// TwinCAT 3 PLC project Untitled1
// ProgramVersion: 3.1.4024.0
// libraries:
//   Tc2_Math, * (Beckhoff Automation GmbH)
//   Tc2_Standard, * (Beckhoff Automation GmbH)
//   Tc2_System, * (Beckhoff Automation GmbH)
//   Tc2_Utilities, * (Beckhoff Automation GmbH)
//   Tc3_Mc3PlanarMotion, * (Beckhoff Automation GmbH)
//   Tc3_Module, * (Beckhoff Automation GmbH)
//   Tc3_Physics, * (Beckhoff Automation GmbH)
//   Tc3_XPlanarUtility, * (Beckhoff Automation GmbH & Co. KG)
//   XboxControllerUtilities, * (Beckhoff Community)
// project tree:
//   DUTs/ Motion_Parameters.TcDUT, Environment_Parameters.TcDUT
//   / PlcTask.TcTTO
//   POUs/Controller/ XboxController.TcPOU
//   POUs/Demo/ Demo.TcPOU
//   POUs/Enviorment/ Environment.TcPOU
//   POUs/ MAIN.TcPOU
//   POUs/Xplanar/Mover Type/ AMP4220.TcPOU, AMP4330.TcPOU
//   POUs/Xplanar/ XPlanarMover.TcPOU
// real-time tasks:
//   TASK Job Task: cycle default, priority 13
//   TASK PlcTask: cycle T#250us, priority 10, ADS port 350
//   TASK XPlanar Task3: cycle T#250us, priority 4, ADS port 351
//   TASK XPlanar Task4: cycle T#250us, priority 6, ADS port 352
//   TASK MC-Task (MET): cycle T#250us, priority 8, ADS port 353
//   TASK MC-Task (MPT): cycle T#10ms, priority 14, ADS port 354
// variable links:
//   XPlanar MC Project/Axes/Mover4220_1 <-> TcCOM Objects/XPlanar/Mover4220_1
//     McToIo/STD <-> InputsFromNC3/NC3ToHW
//   Untitled1/Untitled1 Instance <-> XPlanar MC Project/Axes/Mover4220_1
//     PlcTask Inputs/MAIN.MyMover.Xplanar_Mover.MCTOPLC/ACT <-> McToPlc/ACT
//     PlcTask Inputs/MAIN.MyMover.Xplanar_Mover.MCTOPLC/COORDMODE <-> McToPlc/COORDMODE
//     PlcTask Inputs/MAIN.MyMover.Xplanar_Mover.MCTOPLC/SET <-> McToPlc/SET
//     PlcTask Inputs/MAIN.MyMover.Xplanar_Mover.MCTOPLC/SETONTRACK <-> McToPlc/SETONTRACK
//     PlcTask Inputs/MAIN.MyMover.Xplanar_Mover.MCTOPLC/STD <-> McToPlc/STD
//     PlcTask Outputs/MAIN.MyMover.Xplanar_Mover.PLCTOMC/STD <-> PlcToMc/STD
//   TcCOM Objects/XPlanar/Mover4220_1 <-> XPlanar MC Project/Axes/Mover4220_1
//     OutputsToNC3/HWToNC3 <-> IoToMc/STD

CONFIGURATION Untitled1
    RESOURCE PLC ON TwinCAT3
        TASK PlcTask(INTERVAL := T#250us, PRIORITY := 10);
        PROGRAM MAIN WITH PlcTask : MAIN;
    END_RESOURCE
END_CONFIGURATION

// ---- DUTs/Motion_Parameters.TcDUT
TYPE Motion_Parameters :
STRUCT
	
	
			maxAcceleration					: 		LREAL	:= 15000;			// mm/s^2
		
			maxVelocity						: 		LREAL	:= 500.0;			// mm/s
		
			minVelocity						: 		LREAL	:= -500.0;			// -mm/s
		
			RotationScailing				: 		LREAL 	:= 0.0005; 			// Radians/s^2
		
			CenteringFactor					:		LREAL	:= 0.002;			// Radians/s^2
		
			tiltscailing					:  		LREAL 	:= 0.008; 			// scailing from controller to radians 

END_STRUCT
END_TYPE

// ---- DUTs/Environment_Parameters.TcDUT
TYPE Environment_Parameters :
STRUCT
	
			Friction_coefficient			:  		LREAL 	:= 9.50 ; 			// Frictiton of table
			
			deltaT							:		LREAL	:= 0.00025;			//Cycle time 

END_STRUCT
END_TYPE

// ---- POUs/MAIN.TcPOU
PROGRAM MAIN
VAR
	
MyMover : XplanarMover; // Xplanar Mover

MyController : XboxController; // Xbox Controller

MyEnvironment : Environment; // Xplanar Environment

MyDemo : Demo; // Xplanar Demo 

END_VAR
























VAR
	bRumble : BOOL;  // Set rumble true for haptics based on conditions
END_VAR

Cyclic(); 


MyMover(
// Part number of mover being controlled	
MoverType := 'AMP4220',
Space_Mode := FALSE //Fun time - need to reactivate if set true or false 
); 

MyController(
// Set true if you want haptics and false if you dont	
HapticFeedback := TRUE
);

MyEnvironment(
// Input number of X and Y tiles youre table has
NumberOfXTiles := 4, 
NumberOfYTiles := 3	
);

ACTION Cyclic:
Haptics();

//Initizalization
MyMover.Init( 
bStart := MyController.Start,
Reinit := MyDemo.StartUserControl
);

//Recover 
MyMover.Recover(
bBack := MyController.Reset
); 

//tilt
MyMover.Tilt_Height(
rStick_X := MyController.rStick_X,
rStick_Y := MyController.rStick_Y,
bButton_B := MyController.Button_B,
LBumper := MyController.lBumper,
RBumper	:= MyController.rBumper
);

//X and Y Movement 
MyMover.XYMovement(
lStick_X := MyController.lStick_X, 
lStick_Y := MyController.lStick_Y, 
bButton_A := MyController.Button_A, 
bButton_X := MyController.Button_X, 
bButton_Y := MyController.Button_Y, 
maxXTravel := MyEnvironment.MaxTableXTravel,
minXTravel := MyEnvironment.MinTableXTravel,
maxYTravel := MyEnvironment.MaxTableYTravel,
minYTravel := MyEnvironment.MinTableYTravel,

);

MyMover.Rotation(
LTrigger := MyController.lTrigger,
RTrigger := MyController.rTrigger
);

MyController.takeScreenshot(
bDpad_D := Mycontroller.Dpad_D,
MoverPosition := MyMover.Xplanar_Mover.MCTOPLC.ACT.ActPos
);

MyController.clearScreenshot(
bDpad_U := MyController.Dpad_U,
ClearPosition := MyController.ZeroVector
);

MyController.Haptics(
Rumble := bRumble,
BackTo0Rumble := MyMover.RotationRumble
);

MyEnvironment.Boundry(
MoverTypeWidth 				:= MyMover.TypeWidth, 
MoverTypeLength				:= MyMover.TypeLength 
);

MyMover(
StartDemo := MyDemo.RequestDemo,
DemoNotReady :=  MyDemo.StartUserControl
); 


MyDemo(
ReadyForDemo := MyMover.DemoReady,
bDpad_R := MyController.Dpad_R,
bDpad_L := MyController.Dpad_L,
StopEndFunction := MyMover.ResetDemo,
DemoTable := MyEnvironment.TableType,
//Running := MyMover.FourByThree.Running OR MyMover.TwoByOne.Running,
//Done := MyMover.FourByThree.Done OR MyMover.TwoByOne.Done
);

MyMover.FourByThree(
Start:= MyDemo.StartFourByThree,
Stop := MyDemo.StopFourByThree
);

MyMover.TwoByOne(
Start:= MyDemo.StartTwoByOne,
Stop := MyDemo.StopTwoByOne
);




MyMover(); 
MyController();
MyEnvironment();
MyDemo();
END_ACTION

METHOD Haptics
VAR_INPUT
END_VAR
VAR_OUTPUT
END_VAR
VAR
END_VAR
//When found a rotation point or at a boundry 
IF NOT MyMover.Space_mode THEN // IF space mode is on chnage the way table detection is done
	IF (MyController.Button_A AND MyMover.RotationXPoint AND MyMover.RotationYPoint) 
	OR (MyController.lBumper OR MyController.rBumper) 
	OR ((MyEnvironment.MinTableXTravel + 1 > MyMover.PlanarMoverPos.X) 
	OR (MyEnvironment.MinTableYTravel + 1 > MyMover.PlanarMoverPos.Y) 
	OR (MyEnvironment.MaxTableYTravel - 1 < MyMover.PlanarMoverPos.Y) 
	OR (MyEnvironment.MaxTableXTravel - 1 < MyMover.PlanarMoverPos.X))THEN
		bRumble := TRUE;
	ELSE
		bRumble := FALSE;
	END_IF
ELSE
	//Increase mover detection on boundry
	IF (MyController.Button_A AND MyMover.RotationXPoint AND MyMover.RotationYPoint) 
	OR (MyController.lBumper OR MyController.rBumper) 
	OR (((MyEnvironment.MinTableXTravel + 15) > MyMover.PlanarMoverPos.X) 
	OR ((MyEnvironment.MinTableYTravel + 15) > MyMover.PlanarMoverPos.Y) 
	OR ((MyEnvironment.MaxTableYTravel - 15) < MyMover.PlanarMoverPos.Y) 
	OR ((MyEnvironment.MaxTableXTravel - 15) < MyMover.PlanarMoverPos.X))THEN
		bRumble := TRUE;
	ELSE
		bRumble := FALSE;
	END_IF
END_IF
END_METHOD

END_PROGRAM

// ---- POUs/Xplanar/XPlanarMover.TcPOU
FUNCTION_BLOCK XPlanarMover
VAR_INPUT
	
			MotionParameters			:		Motion_Parameters; // Min-max Motion parameters

			MoverType					: 		STRING(7); //Input what mover is being controlled
			
			Space_mode					:		BOOL; // Space mode ???
			
			StartDemo					:		BOOL; // Change to Demo
			DemoNotReady 				: 		BOOL; //Handeling for end process

END_VAR
VAR_OUTPUT
	
			Xplanar_Mover 				: 		MC_PlanarMover; // Xplanr Mover fb
			moverState					:		MC_Planar_State; // State of mover
			
			TypeWidth					: 		LREAL; //Mover Width  		
			TypeLength					:		LREAL; //Mover Length
			
			PlanarMoverPos				:		MoverVector; // Haptic Handeling
			
			RotationXPoint				:		BOOL; // At rotation point for haptics
			RotationYPoint				:		BOOL; // At rotation point for haptics
			RotationRumble				:		BOOL; // At 0 output for haptics
			
			DemoReady					:		BOOL; // Handshake to start demo
			ResetDemo					:		BOOL; // Hnadshake to stop end demo
			
END_VAR
VAR
	
			stExtOptions				:		ARRAY [1..2]  OF ST_ExternalSetpointGenerationOptions; // External Setpoint options
			cmdFB 						:		ARRAY [1..2]  OF MC_PlanarFeedBack ; //Mover Feedback 
			XpPosition					:		MoverVector; // Commanded mover pos
			MoverPos					:		MoverVector; // Act pos of mover
			ZeroVector 					:		MoverVector; // Zero feed for External Pos

			
			
			EnvironmentParameters		:		Environment_Parameters; // Enviroment parameters like table boundry, fricition coeffecent 
			typeAMP4220					: 		AMP4220; // Mover 4220 decleration	
			typeAMP4330					:		AMP4330; // Mover 4330 decleration
			
		
			//Init Vars
			Run 						:		BOOL; // Run init case	
			DONE						: 		BOOL; // Done running init
			nCase 						: 		SINT := 1; // Case of init
			init_counter				:		INT; // How many times we can try to recover

			
 			//X Y vars
			SumnedForce_X				: 		LREAL; // Calculation of applied force on X
			SumnedForce_Y 				: 		LREAL; // Calculation of applied force on Y
			Mover_acceleration			: 		MoverVector; // Commanded Mover Acc
			friction_force				: 		MoverVector; // Fricition against mover
			SumnedVelocity				: 		MoverVector; // Commanded Velocity after intergation 
			
			
			//Recover Vars
			nRecover					:		SINT := 1; // Case of Recover
			bRecover					: 		BOOL; // Recover mover 
			
			
			//Height Vars
			Height 						: 		LREAL := 2; // Varible in which height is passed
			Left_OSR					: 		R_TRIG; // OSR to make sure a left bumper click is counted a one
			Right_OSR					: 		R_TRIG; // OSR to make sure a right bumper click is counted a one
			Left_Bumer_TON				:		TON; // Timer for incremental lowering 
			Right_Bumper_TON			:		TON; // Timer for incremental rising 
			Smoothing_Left_TON			:		TON; // Timer for smoothing on lowering 
			Smoothing_Right_TON			:		TON; // Timer for smoothing on rising 
			
			//Tilt Vars
			Holding_Contact				:		BOOL; // Holding bool for Button B
			Release_Contact				:		BOOL; // Release bool for holding contact
			Button_B_OSR				: 		R_TRIG; // OSR to make sure a Button B click is counted a one
			nButton						:		INT := 1; // Case for holding contact
			
			//Rotation Vars
			DestinationX				: 		DINT; // Rotation point on X plane
			DestinationY				: 		DINT; // Rotation point on Y plane 
			AtXPoint					: 		BOOL; // At x point on table 
			AtYPoint					: 		BOOL; // At Y point on table 
			MaxPosRot					: 		LREAL; // Max Positive rotation allowed if not at rotation point
			MaxNegRot					: 		LREAL; // Max Negative rotation allowed if not at rotation point
			isintent					: 		BOOL; // mChecking to see if mover is standstill
			Closest90					:		LREAL; // Finding the closest position that is moduled by 90 from actual pos
			MODDED_C					: 		INT; // Modded C value for math check
			PastRot10					: 		BOOL; // Past +- 01 degress check
			Centering_Direction			:		SINT; // Check to see which direction mover needs to center in
			LowerBound 					: 		LREAL; // Lower bound of Centering position
			UpperBound 					: 		LREAL; // Upper bound of Centering position
			Rotation0Rumble				:		BOOL; // Set rumble if rotation goes back to 0
			
			//End Vars
			nEnd						:		SINT := 0; // Start End Procces
			
			//Demo Vars
			
END_VAR
VAR_IN_OUT
END_VAR

Cyclic(); 


	//External Setpint Generator 
	Xplanar_Mover.SetExternalSetpoint( XpPosition, ZeroVector, ZeroVector);

ACTION Cyclic:
//Mover 1 updates
Xplanar_Mover.Update();  // Updating Mopver FB
cmdFB[1].Update(); // Updating Mover feedback
moverState := Xplanar_Mover.MCTOPLC.STD.State; // passing in mover state 
MoverPos := Xplanar_Mover.MCTOPLC.ACT.ActPos; // passing in mover act pos
PlanarMoverPos := Moverpos;
RotationXPoint := AtXPoint;
RotationYPoint := AtYPoint;
RotationRumble := Rotation0Rumble;
typeAMP4220(); // update mover 4220 FB
typeAMP4330(); // Update mover 4330 FB
EndMover();

//Choose varibles to pass based on which mover is called
IF MoverType = 'AMP4220' THEN
	TypeWidth := typeAMP4220.MoverTypeWidth;
	TypeLength := typeAMP4220.MoverTypeLength;
ELSIF MoverType = 'AMP4330' THEN
	TypeWidth := typeAMP4330.MoverTypeWidth;
	TypeLength := typeAMP4330.MoverTypeLength;
END_IF
END_ACTION

METHOD EndMover
VAR_INPUT
	


END_VAR

VAR
	
MoveC_Dyn			:		DynamicConstraint_PathXY;
	
END_VAR

MoveC_Dyn.SetValuesVADJ(500,5000,5000,20000);

IF NOT StartDemo THEN 
	DemoReady := FALSE;
END_IF


IF StartDemo THEN 
	CASE nEnd OF
	
	0:
		//Idle
		IF NOT DemoReady THEN
			nEnd := nEnd + 1;	
		END_IF
	
	1:
		
		//Set function block done bit to false to halt all moves
		Done := FALSE;
		nEnd := nEnd + 1;
		
	2:
	
		IF NOT Done THEN
			nEnd := nEnd + 1;
		ELSE 
			nEnd := 1;
		END_IF
	3:
		
		// Stop the external setpoint generator 
		Xplanar_Mover.StopExternalSetpointGeneration(cmdfb[1]);
		nEnd := nEnd + 1;
		
		
	4:
		
		//Snap mover to 0
		IF MoverPos.c <> 0 THEN
			Xplanar_Mover.MoveC(cmdfb[1],LREAL_TO_INT(Closest90),MoveC_Dyn,0);
			nEnd := nEnd + 1;
		END_IF
		
	5:
	
		//Set demo ready bit 
		DemoReady := TRUE; 
		ResetDemo := FALSE;
		nCase := 1;
		nEnd := 0;
	
	
		
	END_CASE
END_IF
END_METHOD

METHOD FourByThree 
VAR_INPUT
	
	Start				:			BOOL;
	Stop				:			BOOL;

END_VAR
VAR_OUTPUT
	
			Running				:			BOOL; 
			Done				:			BOOL;
			nRecover					:		SINT := 1; // Case of Recover
	
END_VAR
IF Start THEN
//	
END_IF
END_METHOD

METHOD Init
VAR_INPUT
	
	bStart 						: 		BOOL; // Start button on controller
	Reinit						:		BOOL; // Start mover after demo

END_VAR
VAR
	
END_VAR



IF bStart AND NOT StartDemo THEN
	Run := TRUE;
END_IF

IF (Run OR bRecover OR Reinit) AND NOT (init_counter = 3)   THEN
	CASE nCase OF
	1: 
	
		//Reset Mover
		Done := FALSE;
		Xplanar_Mover.Reset(cmdFB[1]);
		nCase := 2;
	
	2:
	
		// Check to see if done with action
		IF cmdFB[1].Done THEN
			nCase := 3; 
		END_IF
		
	3:
	
		// Enable mover
		Xplanar_Mover.Enable(cmdFB[1]);
		nCase := 4;
		
	4:
	
		// Check to see if done with action
		IF cmdFB[1].Done THEN
			nCase := 5;
		END_IF
		
	5:
	
		// Start External Setpoint generator 
		stExtOptions[1].mode := MC_EXTERNAL_SET_POSITION_MODE.Absolute; // Setting up external Setpoint generator
		nCase := 6; 
	
	6:
	
		// If mover is errored then re init 
		IF  MoverState = 5 OR  MoverState = 1 THEN 
			nCase := 1;		
		ELSE 		
			nCase := 7;
		END_IF 
	
	7:
	
		// If mover enabled continue 
		IF MoverState = 3 THEN 
			nCase := 8;
		END_IF
	
	
	8:
		
		// Check to see if done with action
		// Update Positions to real world value before initization of External Setpoint
		IF cmdFB[1].Done  AND NOT cmdFB[1].Busy AND NOT cmdFB[2].Busy  THEN
			XpPosition.y := MoverPos.y; 
			XpPosition.x := MoverPos.x; 
			XpPosition.z := MoverPos.z;
			XpPosition.c := MoverPos.c;
			nCase := 9;
		END_IF
	
	
	9:
	
		// Start External Setpoint Generatior
		Xplanar_Mover.StartExternalSetpointGeneration(cmdFB[1], stExtOptions[1]); 
		nCase := 10; 
		
	10:
	
	// If errored be able to reset 
	IF MoverState = 5 OR  MoverState = 1 THEN
		init_Counter := init_Counter + 1; 
		nCase := 1; 
	ELSE
		Done := TRUE; // Set true to allow for movement 
		Run := FALSE; // Dont call init over again
		bRecover := FALSE; // Dont recover if enabled and ready
		init_counter := 0; // Reset init try's counter
		ResetDemo := TRUE;
	END_IF
		
	END_CASE
END_IF
END_METHOD

METHOD Recover
VAR_INPUT
	
			bBack 							: BOOL ; 

END_VAR
CASE nRecover OF 
	1:
	
		IF Done OR (init_Counter = 3) THEN
			nRecover := nRecover + 1;
		END_IF
	
	2:
	
		IF  MoverState = 5 OR  MoverState = 1 THEN
			Done := FALSE; // Done bit false so no movement can be called	
			nRecover := nRecover + 1; 
		END_IF
		
	3:
	
		//Mapped as reset of mover
		IF bBack = TRUE THEN
			Xplanar_Mover.StopExternalSetpointGeneration(cmdfb[1]);
			nRecover := nRecover + 1; 
		END_IF
		
	4:
		
		nCase := 1; // places in case one of init 	
		bRecover := TRUE; // Calls init of mover
		init_counter := 0; // Resets mover init count 
		nRecover := nRecover + 1; 
	
	5:
	
		nRecover := 1;

END_CASE
END_METHOD

METHOD Rotation : BOOL
VAR_INPUT
	
			LTrigger 					: 		LREAL ; // Left trigger - left rotation
			RTrigger 					: 		LREAL ; // Right Trigger - right rotation 

END_VAR

VAR_OUTPUT
			Rumble 						: 		BOOL; // Set Rumble 
			
END_VAR
IF Done THEN 
	
//Rotation Handeling

		// Find Nearest X rotation point based on act pos
		IF LREAL_TO_INT(MoverPos.X) MOD 120 < 60 THEN
			DestinationX	:= 120 * MODTURNS(MoverPos.X , 120);
		ELSE
			DestinationX	:= 120 * (MODTURNS(MoverPos.X, 120) + 1);
		END_IF
		
		// Find Nearest Y rotation point based on act pos
		IF LREAL_TO_INT(MoverPos.Y) MOD 120 < 60 THEN
			DestinationY	:= 120 * MODTURNS(MoverPos.Y , 120);
		ELSE
			DestinationY	:= 120 * (MODTURNS(MoverPos.Y, 120) + 1);
		END_IF
		
		// Set Boundries for X to not move to edge of table 
		IF DestinationX = 0 THEN
			DestinationX := DestinationX + 120;
		ELSIF DestinationX = 960 THEN
			DestinationX := DestinationX - 120;
		END_IF 	
		
		// Set Boundries for Y to not move to edge of table 
		IF DestinationY = 0 THEN 
			DestinationY := DestinationY + 120;
		ELSIF DestinationY = 720 THEN
			DestinationY := DestinationY - 120;
		END_IF 		
		
		// The direction the mover neds to turn to home to our closest 90 value
		IF Closest90 <= MoverPOs.c THEN
			Centering_Direction := -1; 
		ELSE
			Centering_Direction := 1;
		END_IF
		
		// Set Lower and Upper Bounds
		lowerBound := (Closest90 - 0.3);
		UpperBound := (Closest90 + 0.3);
		
		
		//Checking to make sure Tile is within 1 mm +- of a point that is modulo by 120 and = 0 and then truning a bool true or false
		IF ((LREAL_TO_INT(MoverPos.x) MOD 120) >= 119) OR ((LREAL_TO_INT(MoverPos.x) MOD 120) <= 1)  THEN
			AtXPOint := TRUE; 
		ELSE 
			AtXPoint := FALSE; 
		END_IF
		
		IF ((LREAL_TO_INT(MoverPos.y) MOD 120) >= 119) OR ((LREAL_TO_INT(MoverPos.y) MOD 120) <= 1) THEN
			AtYPOint := TRUE; 
		ELSE
			AtYPoint := FALSE;
		END_IF	
		
		
		//Modded C Value
		//Make sure to not divide by 0 
		IF  MoverPos.c <> 0 THEN
			MODDED_C:=LREAL_TO_INT(MODABS(MoverPos.c,90));
		END_IF	
		
		IF Modded_C <= 45 THEN 
			Closest90 := LREAL_TO_INT(MoverPos.c) - Modded_C;  // find our closet 90
		ELSIF Modded_C >= 46 THEN
			Closest90 := LREAL_TO_INT(MoverPos.c) + ( 90 - Modded_C); // find our closet 90
		END_IF
		
		MaxNegRot := Closest90 - 10; // Our max neg rotation that can happen based off closet 90
		MaxPosRot := Closest90 + 10; // Our max pos rotation that can happen based off closet 90


		//Cant move out of rotation point unless within 10 degress 
		IF (10.1 <= Modded_C)AND (Modded_C <= 79.9) THEN
			PastRot10 := TRUE;
		ELSE 
			PastRot10 := FALSE; 
		END_IF
		
		
		//Endless Rotation 
		IF (AtXPoint AND AtYPoint) AND isintent THEN // If mover is at X and y rotation point and the rotation is intentenal and A button is not pressed
			IF (RTrigger >= 5 AND LTrigger <= 5) THEN // 
				//Negative Rotation
				XpPosition.c := XpPosition.c - ( MotionParameters.RotationScailing * RTrigger);			
			ELSIF LTrigger >= 5 AND RTrigger <= 5 THEN
				//Positive Rotation 
				XpPosition.c := XpPosition.c + (MotionParameters.RotationScailing * LTrigger);
			ELSE 
				 // Do nothing  
			END_IF
		ELSE	
			IF NOT PastRot10 THEN // If A is not pressed and we are not past +- 10 degrees
				//+-10 Rotation Control
				IF LTrigger = 0 AND RTrigger = 0 THEN
		  			(* If both triggers are inactive, move towards 0 (center) gradually *)
		  			IF MoverPos.c > (UpperBound) OR MoverPos.c < (lowerBound) THEN
		  				XpPosition.c := XpPosition.c + (MotionParameters.CenteringFactor * Centering_Direction); 
		  			END_IF
				ELSE
		  			(* If any trigger is active, update the rotation value accordingly *)
		  			XpPosition.c := LIMIT(MaxNegRot, XpPosition.c + (MotionParameters.RotationScailing * LTrigger) + (-1*( MotionParameters.RotationScailing * RTrigger)) , MaxPosRot);
				END_IF
			END_IF
		END_IF
	

		IF LTrigger = 0 AND RTrigger = 0  THEN
			IF MoverPos.c > (UpperBound+ 0.3) OR MoverPos.c < (lowerBound -0.3) THEN
				Rotation0Rumble := FALSE; // Set Rumble 
			ELSE
				Rotation0Rumble := TRUE; // Set Rumble 
		  	END_IF
		END_IF
		

		
		
END_IF
END_METHOD

METHOD Tilt_Height
VAR_INPUT

//Tilt Inputs	
rStick_X 				: LREAL; // Right stick X axis - tilt on B
rStick_Y				: LREAL; // Right stick Y axis - tilit on A
bButton_B 				: BOOL;  // Button B on controller - anti slosh

//Height inputs
LBumper					: 	BOOL;
RBumper					:	BOOL;

END_VAR
VAR_IN_OUT
END_VAR
IF Done THEN 
	

	// Hold down for automatic raise and lowering
	Left_Bumer_TON(IN := LBumper, PT := T#0.25S); 
	Right_Bumper_TON(IN := RBumper, PT := T#0.25S);
	Smoothing_Left_TON(PT := T#0.1S);
	Smoothing_Right_TON(PT := T#0.1S);

	// If timer then activate other then repeat
	IF Left_Bumer_TON.Q THEN
		Smoothing_Left_TON.IN := TRUE AND NOT Smoothing_Left_TON.Q;
	ELSE
		Smoothing_Left_TON.IN := FALSE;		
	END_IF
	
	// If timer then activate other then repeat
	IF Right_Bumper_TON.Q THEN
		Smoothing_Right_TON.IN := TRUE AND NOT Smoothing_Right_TON.Q;
	ELSE
		Smoothing_Right_TON.IN := FALSE;
	END_IF
	
	
	// OSR to make sure only one is seen per click if intention
	Left_OSR(CLK:= LBumper, Q=> ); // OSR for left bumper 
	Right_OSR(CLK:= RBumper, Q=> ); // OSR for right bumper 
	
	// Raise and lowering of mover + implemntation of limits on height
	// Can go negative for holding force 
	IF NOT Holding_Contact THEN
		IF (Left_OSR.Q OR Smoothing_Left_TON.Q) AND Height >= -0.35 THEN 
			Height :=  Height - 0.15; // Decrease Height 
		ELSIF (Right_OSR.Q OR Smoothing_Right_TON.Q) AND Height < 5.0 THEN
			Height := Height + 0.15; // Increase Height 
		ELSE
			Height := Height; // No change 
		END_IF
	ELSE
		Height := 2.0; // Height for anti slosh
	END_IF

	XPPosition.z		:= Height; // Passing in height to Exterenal setpoint generator
	
	
	
	
	
	
	
	
	
	
	
	
	
	
	
	
	Button_B_OSR(CLK := bButton_B, Q => ); // OSR for b button
	
	CASE nButton OF 
	1:
		// Set holding contact true
		IF Button_B_OSR.Q THEN
			Holding_Contact := TRUE;
			Release_Contact := FALSE;			
			nButton := 2;
		END_IF
		
	2:	
	
		// Set release contact true
		IF Button_B_OSR.Q AND Holding_Contact THEN
			Release_Contact := TRUE;
			nButton := 3;
		END_IF
	3:
	
		// Turn off holding contact
		IF Release_Contact THEN
			Holding_Contact := FALSE;
			nButton := 1;
		END_IF
	END_CASE

	

	IF NOT Holding_Contact THEN	
		//A tilt 
		XpPosition.a	:= MotionParameters.tiltscailing * rStick_Y; // Normal a tilt function
		
		//B tilt 	
		XPPosition.b   	:= MotionParameters.tiltscailing * rStick_X; // Normal b tilt function
	ELSE
		IF SumnedVelocity.y > (0.0001) OR SumnedVelocity.y < (-0.0001) THEN // set to 0 if beyond epsilon check 
			XpPosition.a	:=  SumnedVelocity.y * 0.00159681; // a tilt proptional to velocity on y axis
		ELSE
			XpPosition.a	:=  0.0; 
		END_IF
		
		IF SumnedVelocity.x > (0.0001) OR SumnedVelocity.x < (-0.0001) THEN // set to 0 if beyond epsilon check
			XPPosition.b  	:= SumnedVelocity.x * 0.00159681; // b tilt proptional to velocity on x axis
		ELSE
			XpPosition.b 	:=  0.0;
		END_IF
	END_IF

END_IF
END_METHOD

METHOD TwoByOne
VAR_INPUT
	
	Start				:			BOOL;
	Stop				:			BOOL;

END_VAR
VAR_OUTPUT
	
	Running				:			BOOL; 
	Done				:			BOOL;
	
END_VAR
END_METHOD

METHOD XYMovement
VAR_INPUT
	
			lStick_X 					: 		LREAL; // Left stick X axis - X movement of mover
			lStick_Y					: 		LREAL; // LEft stick Y axis - Y movement of mover
			                    	      		
			bButton_A 					: 		BOOL;  // Button A on controller - homing to rotation position
			bButton_X 					: 		BOOL;  // Button X on controller - locking into X movement 
			bButton_Y 					: 		BOOL;	 // Button Y on controller - locking into Y movement
			                    	      		
			maxXtravel          	    : 		LREAL; // Max X travel on table
			minXTravel          	    : 		LREAL; // Min X travel on table
			maxYTravel          	    : 		LREAL; // Max Y travel on table
			minYTravel					: 		LREAL; // Min Y travel on table

END_VAR
VAR
END_VAR
VAR_IN_OUT
END_VAR
IF Done THEN 

	//Imitate driving in space with thrusters
	IF Space_Mode THEN
		EnvironmentParameters.Friction_coefficient := 0.35; // Turn down coeffeint to match space like conditions
		
		//Setting up elastic boundry
		IF XpPosition.x = MinXtravel OR XpPosition.x = MaxXtravel THEN
			SumnedVelocity.X := -1 * SumnedVelocity.X  ;
		END_IF
		
		IF XpPosition.y = MinYtravel OR XpPosition.Y = MaxYtravel THEN
			SumnedVelocity.y := -1 * SumnedVelocity.y  ;
		END_IF
		
		//Change mover acceleration to better adapt to space like conditions 
		Mover_acceleration.x := lStick_X * MotionParameters.maxAcceleration / 500.0;
   		Mover_acceleration.y := lStick_Y * MotionParameters.maxAcceleration / 500.0;	
		
	ELSE
		
		// Normal moving conditions
		// Read the analog stick inputs (x and y) and scale them to control acceleration
    	// Input values are assumed to be in the range [-200, 200] for both x and y axes
    	// Scale them to the range [-max_acceleration, max_acceleration] for acceleration
		Mover_acceleration.x := lStick_X * MotionParameters.maxAcceleration / 200.0;
   		Mover_acceleration.y := lStick_Y * MotionParameters.maxAcceleration / 200.0;
	
	END_IF

	// Is intention to stop moving based on dead zone
	IF (lStick_X < 15 AND lStick_X > -15 ) AND (lStick_Y < 15 AND lStick_Y > -15)THEN
		isintent := TRUE;
	ELSE 
		isintent := FALSE;;
	END_IF


    // If there is no acceleration command, apply friction to reduce velocity
	friction_force.x := -1 * EnvironmentParameters.Friction_coefficient * SumnedVelocity.x;
	friction_force.y := -1 * EnvironmentParameters.Friction_coefficient * SumnedVelocity.y;

	
	// Reduce acceleration based on the friction force
	SumnedForce_X := Mover_acceleration.x + friction_force.x;
	SumnedForce_Y := Mover_acceleration.y + friction_force.y;

	// Update the object's velocity based on the acceleration (INTEGRATING)
	IF NOT bButton_Y THEN // Dont allow for X movement 
		IF 
		SumnedVelocity.x := LIMIT(MotionParameters.minVelocity, SumnedVelocity.x, MotionParameters.maxVelocity) + (SumnedForce_X * EnvironmentParameters.deltaT);
	ELSE
		SumnedVelocity.x := 0;
	END_IF
	
	IF NOT bButton_X THEN // Dont allow for Y movement 
		SumnedVelocity.y := LIMIT(MotionParameters.minVelocity, SumnedVelocity.y, MotionParameters.maxVelocity) + (SumnedForce_Y * EnvironmentParameters.deltaT);
	ELSE
		SumnedVelocity.Y := 0;
	END_IF
	

	// Move to Nearest Rotation point
	// Go to nearest X point
	IF bButton_A AND MoverPos.X < DestinationX THEN
		XpPosition.X := XpPosition.X + ( 40 * EnvironmentParameters.deltaT );
	ELSIF bButton_A AND MoverPos.X > DestinationX THEN
		XpPosition.X := XpPosition.X -( 40 * EnvironmentParameters.deltaT );
	END_IF;
	
	// Go to nearst Y point 
	IF bButton_A AND MoverPos.Y < DestinationY THEN
		XpPosition.Y := XpPosition.Y + ( 40 * EnvironmentParameters.deltaT );
	ELSIF bButton_A AND MoverPos.Y > DestinationY THEN
		XpPosition.Y := XpPosition.Y -( 40 * EnvironmentParameters.deltaT );
	END_IF;
	
	IF NOT PastRot10 THEN // Dont let mover out of rotation if its passed -+10 degrees
		// Update the object's position based on the velocity(INTEGRATING)	
		XpPosition.x		:= LIMIT(minXTravel, XpPosition.x + ((SumnedVelocity.x) * EnvironmentParameters.deltaT ) ,maxXTravel);
		XpPosition.y		:= LIMIT(minYTravel, XpPosition.y + ((SumnedVelocity.y) * EnvironmentParameters.deltaT ) ,maxYTravel);
	END_IF
	
END_IF
END_METHOD

END_FUNCTION_BLOCK

// ---- POUs/Xplanar/Mover Type/AMP4220.TcPOU
FUNCTION_BLOCK AMP4220 
VAR_INPUT
END_VAR
VAR_OUTPUT
	
			MoverTypeWidth 				: 		LREAL := 56.5; // Mover Width/2 in mm
			MoverTypeLength				: 		LREAL := 56.5; // Mover Length/2 in mm 

END_VAR
VAR
END_VAR

END_FUNCTION_BLOCK

// ---- POUs/Xplanar/Mover Type/AMP4330.TcPOU
FUNCTION_BLOCK AMP4330 
VAR_INPUT
END_VAR
VAR_OUTPUT
	
			MoverTypeWidth 				: 		LREAL := 77.5; // Mover Width/2 in mm
			MoverTypeLength				: 		LREAL := 77.5; // Mover Length/2 in mm 

END_VAR
VAR
END_VAR

END_FUNCTION_BLOCK

// ---- POUs/Controller/XboxController.TcPOU
FUNCTION_BLOCK XboxController
VAR_INPUT
	
			HapticFeedback				:		BOOL; // Haptic feedback enable bit		

END_VAR
VAR_OUTPUT
	
			XboxController				: 		FB_Xbox_Controller(NetID := '', iControllerNumber := 1); // Xbox Controller Decleration 
			bIsConnected   				:  		ARRAY [1..2] OF BOOL; // Controller conection validated 

			Start 						:       BOOL; // Start Buttom
			Reset 						:       BOOL; // Reset Button
			Button_A            		:       BOOL; // Button A
			Button_B                 	:       BOOL; // Button B
			Button_X             		:       BOOL; // Button X
			Button_Y                    :       BOOL; // Button Y
			Dpad_U	                    :       BOOL; // Dpad UP
			Dpad_D	                    :       BOOL; // Dpad Down
			Dpad_R	                    :       BOOL; // Dpad UP
			Dpad_L	                    :       BOOL; // Dpad Down
			lBumper	                    :       BOOL; // Left Bumper
			rBumper	                    :       BOOL; // Right Bumper
			lTrigger                    :       LREAL; // Left Trigger
			rTrigger                    :       LREAL; // Right Trigger
			lStick_Y	                :       LREAL; // Left Stick Y axis
			lStick_X	                :       LREAL; // Left Stick X axis
     		rStick_Y	                :       LREAL; // Right Stick Y axis
     		rStick_X	                :       LREAL; // Right Stick X axis
			
			ZeroVector					:		MoverVector; // Zero Vector 
			
END_VAR
VAR    
	
			Open_Controller_Service		:		NT_StartProcess; // Open ADS server for controller
			RUN							:		BOOL := TRUE; // Run service 
			
			
			//Take Screenshot vars
			TakeScreenshot_OSR			: 		R_TRIG; // OSR to make sure a Dpad Down click is counted a one
			ClearScreenshot_OSR			: 		R_TRIG; // OSR to make sure a Dpad Up click is counted a one
			Captured_Positions			:		ARRAY [0..9] OF MoverVector; // Array of Positions
			Position_index				:		INT; //Indexing through Positions array

			
			//Haptic Feed Back
			HapticTimerMedium			:		TON; // Haptics feedback timer for longer duration

END_VAR

Cyclic();

METHOD clearScreenshot 
VAR_INPUT
	
			bDpad_U 					: 		BOOL; // Dpad Up on controller 
			ClearPosition				:		MoverVector ; // Mover Vector 


END_VAR
ClearScreenshot_OSR(CLK := bDpad_U, Q => );

IF ClearScreenshot_OSR.Q THEN
	Captured_Positions[Position_index] := ClearPosition ;
	Position_index := Position_index + 1;
END_IF

IF Position_index = 10 THEN
	Position_index := 0;
END_IF
END_METHOD

ACTION Cyclic:
XboxController.Cycle(); // Xbox Controller FB cycle 

mapping(); // Call mapping of Controller

init(); // Call init of controller




bIsConnected[1] := XboxController.P_Status.bConnected; // Is controller Connected
END_ACTION

METHOD Haptics 
VAR_INPUT
	
				Rumble 					:	 	BOOL; // Set Rumble 
				BackTo0Rumble			:		BOOL; // Set rumble if mover hits 0
			
END_VAR
VAR 
END_VAR

//Haptic Feedback Duration
HapticTimerMedium(IN :=BackTo0Rumble, PT := T#0.5S);

//Haptic FeedBack
IF HapticfeedBack = TRUE THEN
//When back to a C value that can be moduloed by 90 and = 0 
	IF BackTo0Rumble THEN
		IF (HapticTimerMedium.IN AND NOT HapticTimerMedium.Q) OR Rumble THEN
			XboxController.SetRumble(0,100);
		ELSE
			XboxController.SetRumble(0,0);
		END_IF
	END_IF	
END_IF
END_METHOD

METHOD Init
VAR_INPUT
END_VAR
VAR
			Busy						:		BOOL;
			ERR							:		BOOL;
			ErrID						:		UDINT;
			nRecover					:		SINT := 1; // Case of Recover
END_VAR
//Open Ads Controller Service on start up

IF NOT bIsConnected[1] THEN
	IF RUN = TRUE THEN 
	Open_Controller_Service(
		NETID:='' , 
		PATHSTR:='C:\Program Files\Beckhoff Community\TwinCAT Xbox Controller Service\ADS-Controller-Server.exe' , 
		DIRNAME:= 'C:\Program Files\Beckhoff Community\TwinCAT Xbox Controller Service', 
		COMNDLINE:='start ADS-Controller-Server.exe', 
		START:= TRUE , 
		TMOUT:= T#5S , 
		BUSY=> BUSY , 
		ERR=> ERR , 
		ERRID=> ERRID );
	END_IF
END_IF
END_METHOD

ACTION Mapping:




// Button Mapping
//Mapping from Controller instance to PLC vars
Start 				:= XboxController.P_Buttons.bStart; 
Reset 				:= XboxController.P_Buttons.bBack;
Button_A 			:= XboxController.P_Buttons.bA_Button;
Button_B 			:= XboxController.P_Buttons.bB_Button;
Button_X 			:= XboxController.P_Buttons.bX_Button;
Button_Y 			:= XboxController.P_Buttons.bY_Button;
Dpad_U	 			:= XboxController.P_Buttons.DPad.bUp;
Dpad_D	 			:= XboxController.P_Buttons.DPad.bDown;
Dpad_R	 			:= XboxController.P_Buttons.DPad.bRight;
Dpad_L	 			:= XboxController.P_Buttons.DPad.bLeft;
lBumper	 			:= XboxController.P_Buttons.bLeft_Shoulder;
rBumper	 			:= XboxController.P_Buttons.bRight_Shoulder;
lTrigger			:= XboxController.P_Left_Trigger;
rTrigger			:= XboxController.P_Right_Trigger;
lStick_Y			:= XboxController.P_Left_Joystick.fY;
lStick_X			:= XboxController.P_Left_Joystick.fX;
rStick_Y			:= XboxController.P_Right_Joystick.fY;
rStick_X			:= XboxController.P_Right_Joystick.fX;
END_ACTION

METHOD takeScreenshot : BOOL
VAR_INPUT
	
			bDpad_D 					: 			BOOL ; // Dpad Down on controller
			MoverPosition				:			MoverVector; // Mover Position

END_VAR
TakeScreenshot_OSR(CLK := bDpad_D, Q => );

IF TakeScreenshot_OSR.Q THEN
	Captured_Positions[Position_index] :=  MoverPosition;
	Position_index := Position_index + 1;
END_IF

IF Position_index = 10 THEN
	Position_index := 0;
END_IF
END_METHOD

END_FUNCTION_BLOCK

// ---- POUs/Enviorment/Environment.TcPOU
FUNCTION_BLOCK Environment
VAR_INPUT

			NumberOfXTiles				: 		INT; // Number of X tiles in a System
			NumberOfYTiles				: 		INT; // Number of Y tiles in a System	

END_VAR
VAR_OUTPUT
	
			MaxTableYTravel 			: 		LREAL ; // Max Y travel of mover
			MaxTableXTravel 			: 		LREAL ; // Max X travel of mover
		             
			MinTableYTravel 			: 		LREAL ; // Min Y travel of mover
			MinTableXTravel 			:		LREAL ; // Min X travel of mover
			
			TableType					:		STRING(3); // Table Demo Type 

END_VAR
VAR
	
			Buffer						: 		INT := 5; // Buffer space 
			RotationDisplacement		:		LREAL; // Rotation displacemnt caused by mover   

END_VAR

METHOD Boundry 
VAR_INPUT
	
			MoverTypeWidth 				: 		LREAL; // Movers Width/2
		    MoverTypeLength				: 		LREAL; // Movers Length/2
	
END_VAR 
VAR 
END_VAR
RotationDisplacement :=  (MoverTypeWidth) * SIN(0.1745); // Calculate Rotation displacemnt of Mover


MaxTableYTravel := (NumberOfYTiles * 240) - MoverTypeWidth  - Buffer - RotationDisplacement ; // Calculate Max Y travel of Mover
MaxTableXTravel := (NumberOfXTiles * 240) - MoverTypeLength - Buffer - RotationDisplacement; // Calculate Max X travel of Mover
		
MinTableYTravel :=  MoverTypeWidth   + Buffer + RotationDisplacement; // Calculate Min Y travel of Mover
MinTableXTravel :=  MoverTypeLength  + Buffer + RotationDisplacement; // Calculate Min X travel of Mover


IF NumberOfXTiles = 2 AND NumberOfYTiles = 1 THEN
	TableType := '2x1'; // 2x1 demo table
ELSIF NumberOfXTiles = 4 AND NumberOfYTiles = 3 THEN
	TableType := '4x3'; // 4x3 demo table 
ELSE
	TableType := 'NaN'; // Not a demo table supported 
END_IF
END_METHOD

METHOD Forces 
VAR_INPUT
END_VAR
END_METHOD

END_FUNCTION_BLOCK

// ---- POUs/Demo/Demo.TcPOU
FUNCTION_BLOCK Demo 
VAR_INPUT
	
			DemoTable					: 		STRING(3); // Demo table type 
			bDpad_R						: 		BOOL;	// Dpad Right for starting the demo 
			bDpad_L						: 		BOOL; // Dpad Left to end demo 
			ReadyForDemo				: 		BOOL; // Handhske varible telling to start demo
			DemoStarting				:		BOOL; // Handshake to stop End Demo function
			StopEndFunction				:		BOOL; // Stop End function
			Running						:		BOOL; 
			Done						:		BOOL; 

END_VAR
VAR_OUTPUT
	
			RequestDemo					:		BOOL; // Handhske varible asking to start demo
			StartUserControl 			:		BOOL; // Varible to give user control of mover again
			StartTwoByOne				:		BOOL; 
			StopTwoByOne				:		BOOL;
			StartFourByThree			:		BOOL; 
			StopFourByThree				:		BOOL;
			nRecover					:		SINT := 1; // Case of Recover

END_VAR
VAR

	
			DemoStart					:			BOOL; // start the demo
			StopDemo					:			BOOL;
			End							:			BOOL;// Simuylate demo end 
		
END_VAR


IF bDpad_R THEN //Link to Controller
	DemoStart := TRUE;
	StopDemo := FALSE;
ELSIF bDpad_L THEN
	DemoStart := FALSE;
	StopDemo := TRUE; 
END_IF

IF DemoStart THEN 
	RequestDemo := TRUE;
	IF ReadyForDemo THEN
		IF DemoTable = '2x1' THEN
			StartTwoByOne := TRUE; 
		ELSIF DemoTable = '4x3' THEN
			StartFourByThree := TRUE;
		ELSIF DemoTable = 'NaN' THEN
			//Do Nothing 
		END_IF
	END_IF
ELSE 
	RequestDemo := FALSE;
END_IF



IF StopDemo THEN 
	IF Running OR Running THEN
		IF DemoTable = '2x1' THEN
			StopTwoByOne := TRUE; 
		ELSIF DemoTable = '4x3' THEN
			StopFourByThree := TRUE;
		ELSIF DemoTable = 'NaN' THEN
			//Do Nothing 
		END_IF
	END_IF
END_IF

IF Done THEN
	StopDemo := FALSE;
	RequestDemo := FALSE;
	StartUserControl := TRUE;
	IF StopEndFunction THEN
		StartUserControl := FALSE;
	END_IF
END_IF

END_FUNCTION_BLOCK
